Fanuc KAREL source: ko00036.KL

-- PROVISIONAL review KL for V1013-1; original PC SHA256 1ed15bb0a7c460934d59fabcfb5cd67f8e8c69dfecb87d2d1ecb30a9651589f6
-- Incomplete behavior may be omitted. Consult companion uncertainty JSON. Do not deploy.
PROGRAM KO00036
%NOLOCKGROUP
BEGIN
  -- UNRESOLVED_PC offsets 5-12; opcodes 9D,23
  -- UNRESOLVED_PC offsets 17-66; opcodes 27,27,49,7E,AD,22,1C,22,31,7E,4A
  -- UNRESOLVED_PC offsets 71-75; opcodes 7F
END KO00036
